FUNCTION TryConvert_ULINT_TO_LINT : BOOL
VAR_INPUT
	in : ULINT;
	out : REFERENCE TO LINT;
END_VAR

IF in > DatatypeLimits.MAX_VALUE_OF_ULINT_WHICH_CAN_BE_HELD_IN_A_LINT THEN
	RETURN;
END_IF

out := ULINT_TO_LINT(in);
TryConvert_ULINT_TO_LINT := TRUE;

END_FUNCTION

(* stored: Version 1.1.0.1, ProductVersion 3.1.4024.12
   POU TryConvert_ULINT_TO_LINT: Id {272ff5f8-42f2-4683-a3dd-42e1f0a036aa}, SpecialFunc None *)
